{attribute 'no_explicit_call' := 'do not call this function block directly'} 
FUNCTION_BLOCK SequentialTaskExecutor EXTENDS ToolkitObject IMPLEMENTS IAbortableProcess
VAR
	_ClassName : STRING := __POUNAME();

	_Tasks : List(POINTER_TYPE.OBJECT_POINTER); // of POINTER TO Task  
	
	_ContinueOnTaskError : BOOL;

	_Busy : BOOL;
	_AbortRequested : BOOL;
	_Aborted : BOOL;
	_Error : BOOL;
	_ErrorMessage : ERROR_MESSAGE;
	_AbortReason : ERROR_MESSAGE;
END_VAR

{attribute 'monitoring' := 'call'}
{attribute 'OPC.UA.DA.Property' := '1'}
{attribute 'OPC.UA.DA.Access' := '1'}
PROPERTY FINAL Aborted : BOOL
GET
Aborted := _Aborted;
END_GET
END_PROPERTY

{attribute 'monitoring' := 'call'}
{attribute 'OPC.UA.DA.Property' := '1'}
{attribute 'OPC.UA.DA.Access' := '1'}
PROPERTY AbortReason : REFERENCE TO ERROR_MESSAGE
GET
AbortReason REF= _AbortReason;
END_GET
END_PROPERTY

METHOD AddTask
VAR_INPUT
	task : REFERENCE TO Task; // instance should be managed by external logic
END_VAR
IF NOT __ISVALIDREF(task) THEN
	RETURN;
END_IF

_Tasks.Append(ADR(task));
END_METHOD

{attribute 'monitoring' := 'call'}
{attribute 'OPC.UA.DA.Property' := '1'}
{attribute 'OPC.UA.DA.Access' := '1'}
PROPERTY FINAL Busy : BOOL
GET
Busy := _Busy;
END_GET
END_PROPERTY

{attribute 'monitoring' := 'call'}
PROPERTY ClassName : STRING
GET
ClassName := _ClassName;
END_GET
END_PROPERTY

METHOD ClearInactiveTasks
VAR
	i : DINT;
	task : POINTER TO Task;
END_VAR
FOR i := _Tasks.Count - 1 TO 0 BY -1 DO
	IF i = 0 THEN
		task := _Tasks.Get(0);
		
		IF task^.State = TASK_STATE.EXECUTING OR_ELSE task^.State = TASK_STATE.ABORTING THEN
			CONTINUE;			
		END_IF
	END_IF
	
	_Tasks.RemoveAt(i, FALSE);
END_FOR
END_METHOD

{attribute 'monitoring' := 'call'}
{attribute 'OPC.UA.DA.Property' := '1'}
{attribute 'OPC.UA.DA.Access' := '1'}
PROPERTY FINAL ContinueOnTaskError : BOOL
GET
ContinueOnTaskError := _ContinueOnTaskError;
END_GET
SET
_ContinueOnTaskError := ContinueOnTaskError;
END_SET
END_PROPERTY

{attribute 'monitoring' := 'call'}
{attribute 'OPC.UA.DA.Property' := '1'}
{attribute 'OPC.UA.DA.Access' := '1'}
PROPERTY FINAL Error : BOOL
GET
Error := _Error;
END_GET
END_PROPERTY

{attribute 'monitoring' := 'call'}
{attribute 'OPC.UA.DA.Property' := '1'}
{attribute 'OPC.UA.DA.Access' := '1'}
PROPERTY FINAL ErrorMessage : REFERENCE TO ERROR_MESSAGE
GET
ErrorMessage REF= _ErrorMessage;
END_GET
END_PROPERTY

METHOD Execute 
VAR
	task : POINTER TO Task;
	taskManagerAbortMessage : ERROR_MESSAGE := "TaskManager aborted with reason: ";
END_VAR
START:

IF NOT Busy OR_ELSE _Tasks.Count = 0 THEN
	RETURN;
END_IF

task := _Tasks.Get(0);

__TRY
	CASE task^.State OF
		TASK_STATE.EXECUTING:
			IF _AbortRequested THEN
				_AbortRequested := FALSE;
				
				IF task^.RequestAbort(TRUE) THEN
					task^.State := TASK_STATE.ABORTED;
				ELSE
					RETURN;
				END_IF
			ELSE
				IF task^.Execute(FALSE) THEN
					task^.State := TASK_STATE.DONE;
				ELSE
					RETURN;
				END_IF		
			END_IF

			_Tasks.Remove(task, FALSE);
							
		TASK_STATE.ABORTING:
			IF task^.RequestAbort(FALSE) THEN
				task^.State := TASK_STATE.ABORTED;
				
				_Tasks.Remove(task, FALSE);
			ELSE
				RETURN;
			END_IF
		ELSE
			task^.AbortReason := "";
			task^.ErrorMessage := "";
			
			IF task^.Execute(TRUE) THEN
				task^.State := TASK_STATE.DONE;

				_Tasks.Remove(task, FALSE);
			ELSE
				RETURN;
			END_IF
	END_CASE	
	
	_Tasks.Remove(task, FALSE);	
__CATCH
	task^.ErrorMessage := ExceptionHelper.LastException.ToString(FALSE);
	task^.State := TASK_STATE.ERROR;
	
	_Tasks.Remove(task, FALSE);

	IF NOT ContinueOnTaskError THEN
		setError(ExceptionHelper.LastException.ToString(FALSE));		
		ExceptionHelper.LastException.Throw();
	END_IF	
__ENDTRY

JMP START;
END_METHOD

METHOD RequestAbort
VAR_INPUT 
	reason : ERROR_MESSAGE;
END_VAR
VAR
	task : POINTER TO Task;
END_VAR
IF Busy THEN	
	_AbortReason := reason;
	
	IF _Tasks.Count > 0 THEN
		task := _Tasks.Get(0);
		
		IF task^.State = TASK_STATE.EXECUTING THEN
			_AbortRequested := TRUE;
			RETURN;
		END_IF
	END_IF

	setAborted();
END_IF
END_METHOD

METHOD PRIVATE setAborted
_Busy := FALSE;
_AbortRequested := FALSE;
_Aborted := TRUE;
_Error := FALSE;
END_METHOD

METHOD PRIVATE setBusy
_Busy := TRUE;
_AbortRequested := FALSE;
_Aborted := FALSE;
_Error := FALSE;
END_METHOD

METHOD PRIVATE setError
VAR_IN_OUT CONSTANT
	errorMessage : ERROR_MESSAGE;
END_VAR
_Busy := FALSE;
_AbortRequested := FALSE;
_Aborted := FALSE;
_Error := TRUE;

IF __ISVALIDREF(errorMessage) THEN
	_ErrorMessage := errorMessage;
END_IF
END_METHOD

METHOD Start
IF Busy THEN
	//exceptionFactory.ThrowException(__POSITION(), "Task manager in aborting state", __POUNAME(), ClassName, CurrentNamespace.Name, __POSITION()).Throw();
END_IF

_ErrorMessage := "";
_AbortReason := "";
setBusy();

Start := TRUE;
END_METHOD

END_FUNCTION_BLOCK

(* stored: Version 1.1.0.1
   POU SequentialTaskExecutor: Id {b15464c1-820f-419b-b833-3fb448a1642b}, SpecialFunc None
   Folder Service members: Id {71a6050a-b35d-4e7f-986a-e3c197a59e46}
   Property Aborted: Id {48dd5883-38e1-4ed7-ac45-8890af864301}
   Get Get: Id {a7f13221-4dea-4dcf-aac5-2e6806496d6b}
   Property AbortReason: Id {8143b43b-4f72-45e8-a647-e71b760d3a0b}
   Get Get: Id {8f48fafa-3c4f-4f36-8ac2-ee53b26f3210}
   Method AddTask: Id {1ddc06dd-e791-40bd-9793-0273ac58e922}
   Property Busy: Id {51046490-29bc-409e-b14e-0bd500ceb597}
   Get Get: Id {744d1fb6-8734-4c73-95c3-55013a307b36}
   Property ClassName: Id {6a98787a-71c6-4478-a0d2-fdfcc0bde94d}
   Get Get: Id {4d0c9db1-17bc-492e-b71e-b2d8c7344182}
   Method ClearInactiveTasks: Id {d47d46b3-a29c-4bba-b2d4-d0048167b63a}
   Property ContinueOnTaskError: Id {7ccbd4cb-8125-4f85-b946-5e096c4897ba}
   Get Get: Id {9ffbc127-4897-4527-93e5-33764300eab9}
   Set Set: Id {4545a0f9-28c4-4e12-972c-12412df0f15a}
   Property Error: Id {ae1bbc34-02a9-4708-b23e-b30267b5cc75}
   Get Get: Id {de9267df-4291-4d77-9769-cddbcc7e4364}
   Property ErrorMessage: Id {d2525150-ab0c-411c-8044-fe8044240f66}
   Get Get: Id {69e8e66e-480f-447d-924a-6931208b1734}
   Method Execute: Id {dd0b06c8-bb70-443d-82d8-5a8f59198530}
   Method RequestAbort: Id {0f00df1e-9306-4979-b0c6-a3618c357788}
   Method setAborted: Id {21449bbc-1a0e-417b-b51e-95651b1a159c}
   Method setBusy: Id {d2776870-60b8-457b-9196-0a0f6d87b360}
   Method setError: Id {d3cf674b-3dd0-49f4-9e69-c74490bbda41}
   Method Start: Id {fe085021-b483-439f-92c4-c87b89e49ff7} *)
